{attribute 'TcGenerated'}
{attribute 'no-analysis'}
{attribute 'linkalways'}
// This function has been automatically generated from the project information.
VAR_GLOBAL CONSTANT
    {attribute 'const_non_replaced'}
    stLibVersion_LCLS_General : ST_LibVersion := (iMajor := 2, iMinor := 13, iBuild := 0, iRevision := 0, nFlags := 1, sVersion := '2.13.0');
END_VAR

(* stored: Version 1.1.0.1
   GVL Global_Version: Id {906e4061-9e6e-442c-b3fd-3984f80a7628} *)
